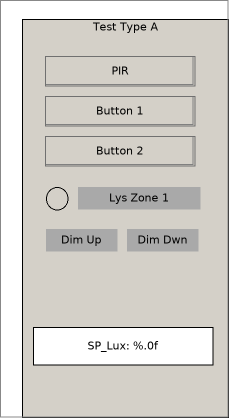
VISUALIZATION Visualization  // 229x418
    RoundedRectangle (22,19 207x399), "Test Type A"
    Button (45,56 150x30), "PIR"
        tap P_Test_TypeA.bPIR
    Rectangle (33,327 180x38), "SP_Lux: %.0f", text variable: P_Test_TypeA.fLuxZone1
    Button (45,96 150x30), "Button 1"
        tap P_Test_TypeA.bButtonZone1
    Button (45,136 150x30), "Button 2"
        tap P_Test_TypeA.bButtonZone2
    Ellipse (46,187 22x23), colour toggle: P_Test_TypeA.bOnZone1
    Rectangle (78,187 122x22), "Lys Zone 1"
    Rectangle (46,229 71x22), "Dim Up", colour toggle: P_Test_TypeA.bDimUp
    Rectangle (127,229 71x22), "Dim Dwn", colour toggle: P_Test_TypeA.bDimDwn
END_VISUALIZATION

(* stored: Version 1.1.0.1
   Visu Visualization: Id {d90fbb08-585d-4679-acf1-1b0da5a9dbeb} *)
